// TIA Portal V18 export
TYPE "RCS_SysAlarmWarning_V1"
   STRUCT
      ON : Bool;   // On Status / Na Stav
      ACK : Bool;   // Acknowledg
      Reset : Bool;
      ImmediatelyStop : Bool;   // Process Immediately Stop / Spracovať Okamžite Zastavte
      CycleStop : Bool;   // Process Cycle Stop / Zastavenie cyklu procesu
   END_STRUCT;
END_TYPE
